Omron CX-Programmer project NewProject (CX-Programmer 9.81)

# PLC Sessao_31_03_2026_Exercicio: CP1L-E EM

## Global symbols (name address type ; comment)
0.00 BOOL  ; Botao Start
0.01 BOOL  ; Temporizador 1
0.02 BOOL  ; Flag do Temporizador 1
0.03 BOOL  ; Botao Stop
0.04 BOOL  ; Botao Start
0.05 BOOL  ; Botao Start 1
0.06 BOOL  ; Botao de Emergencia 2
0.07 BOOL  ; Botao Stop 1
0.08 BOOL  ; Flag do Temporizador 1
0.09 BOOL  ; Botao de Start Esquerdo
0.10 BOOL  ; Botao de Start Direito
0.11 BOOL  ; Temporizador
100 CHANNEL  ; Temporizador
100.00 BOOL  ; Contactor
100.01 BOOL  ; Lampada 2
100.02 BOOL  ; Lampada 3
100.03 BOOL  ; Lampada 4
100.04 BOOL  ; Bobina do Rele
100.05 BOOL  ; Bobina do Motor 1
100.06 BOOL  ; Bobina do Motor 2
100.07 BOOL  ; Temporizador
500 CHANNEL  ; Temporizador 1
T0001 BOOL  ; Flag do Temporizador 1

## Program NewProgram1 (cyclic task 0)
Local symbols
Flag_T1 T0001 BOOL  ; Flag do temporizador 1
KM1 100.00 BOOL  ; Contactor
T_1 1 NUMBER  ; Temporizador 1
Tempo_T1 #55 NUMBER  ; Tempo do temporizador 1
b_start 0.00 BOOL  ; Botao Start
etapa_0 2.00 BOOL  ; Etapa 0 do Grafcet
etapa_1 2.01 BOOL  ; Etapa 1 do Grafcet

### Section Exercicio_1

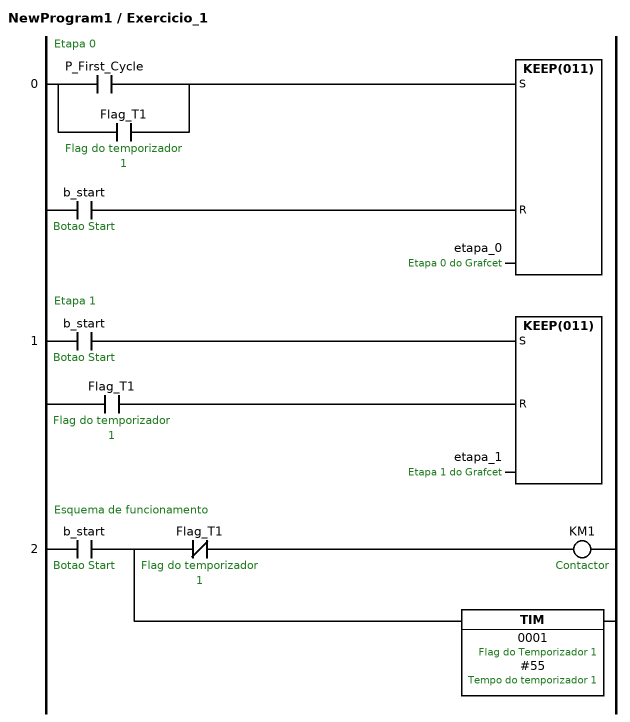
; rung 0: Etapa 0
LD P_First_Cycle
OR Flag_T1  ; Flag do temporizador 1
LD b_start  ; Botao Start
KEEP(011) etapa_0  ; Etapa 0 do Grafcet
; rung 1: Etapa 1
LD b_start  ; Botao Start
LD Flag_T1  ; Flag do temporizador 1
KEEP(011) etapa_1  ; Etapa 1 do Grafcet
; rung 2: Esquema de funcionamento
LD b_start  ; Botao Start
OUT TR0
ANDNOT Flag_T1  ; Flag do temporizador 1
OUT KM1  ; Contactor
LD TR0
TIM 0001 #55  ; Tempo do temporizador 1, Flag do Temporizador 1

### Section END
; rung 0
END(001)